// TwinCAT 3 PLC project Untitled1
// ProgramVersion: 3.1.4022.7
// libraries:
//   Tc2_ModbusSrv, * (Beckhoff Automation GmbH)
//   Tc2_Standard, * (Beckhoff Automation GmbH)
//   Tc2_System, * (Beckhoff Automation GmbH)
//   Tc3_Module, * (Beckhoff Automation GmbH)
// project tree:
//   / PlcTask.TcTTO (not stored)
//   POUs/ MAIN.TcPOU
// real-time tasks:
//   TASK PlcTask: cycle T#10ms, priority 20, ADS port 350

// ---- POUs/MAIN.TcPOU
PROGRAM MAIN
VAR
	fbReadInputs: FB_MBReadInputs;
	DataReadInput	:	BYTE;
	bRead	:	BOOL;
	
	binput1		AT%IX0.0	:	BOOL;
	binput2		AT%IX0.1	:	BOOL;
	binput3		AT%IX0.2	:	BOOL;
	binput4		AT%IX0.3	:	BOOL;
	binput5		AT%IX0.4	:	BOOL;
	binput6		AT%IX0.5	:	BOOL;
	binput7		AT%IX0.6	:	BOOL;
	binput8		AT%IX0.7	:	BOOL;

END_VAR

fbReadInputs(
	sIPAddr:='', 
	nTCPPort:= 502, 
	nUnitID:= 255, 
	nQuantity:= 8, 
	nMBAddr:=0, 
	cbLength:= SIZEOF(DataReadInput), 
	pDestAddr:= ADR(DataReadInput) , 
	bExecute:= bRead, 
	tTimeout:= T#5S, 
	bBusy=> , 
	bError=> , 
	nErrId=> , 
	cbRead=> );
	
	DataReadInput.0;		DataReadInput.1;		DataReadInput.2;		DataReadInput.3;		DataReadInput.4;
	DataReadInput.5;		DataReadInput.6;		DataReadInput.7;		DataReadInput.8;

END_PROGRAM
